FUNCTION alg_a_Dstartled : BOOL
VAR_INPUT
	state: STATE;
END_VAR

alg_a_Dstartled := alg_M_Distributing_a_Dstartled(state);

END_FUNCTION

(* stored: Version 1.1.0.1, ProductVersion 3.1.4022.18
   POU alg_a_Dstartled: Id {176ce68c-9807-416d-a7be-a641f4fd1528}, SpecialFunc None *)
